(* PLC project static_torsion.project, CODESYS CODESYS V3.5 SP17 Patch 3 *)
(* stored: creationDateTime 1970-01-01T00:00:00, modificationDateTime 2026-06-22T15:12:39.4699931 *)

TYPE WORD_TO_STRUCT : UNION
  _PDI : PDI;
  _PDQ : PDQ_OLD;
  _S_CTRL : S_CTRL;
  _S_STATE : S_STATE;
  _WORD : WORD;
END_UNION;
END_TYPE
